FUNCTION_BLOCK FB_SequenceCONVEY_RETRACT EXTENDS FB_SequenceBase



VAR_IN_OUT
	devices: ST_POPComponents;
END_VAR

METHOD FB_init : BOOL
VAR_INPUT
	bInitRetains : BOOL; // if TRUE, the retain variables are initialized (warm start / cold start)
	bInCopyCode : BOOL;  // if TRUE, the instance afterwards gets moved into the copy code (online change)
	
	
END_VAR
(*
		Here we set the order of things to command, what the commands should be, and also how much time to allow during and between steps
		Every component listed below becomes 'Enabled' at each step
*)
sSequenceName:= 'POP Conveyor Reverse Sequence';
sSequenceDescription := 'Performs the full reverse series of actions (starting with lifting movement and followed by static conveyors';
bSequentional_1_Flood_0 := TRUE;
END_METHOD

METHOD populateSteps : ST_SequenceStep
VAR_INPUT
	
END_VAR
(*
		Here we set the order of things to command, what the commands should be, and also how much time to allow during and between steps
		Every component listed below becomes 'Enabled' at each step
*)

Step1.Device := devices.fbLinAct_POP1;
Step1.Command := E_DeviceState.RETRACTED;
Step1.StepMinDuration := T#0S; 
Step1.DelayUntilNextStep := T#0S;
Step1.WaitForAction := FALSE;
aSequenceSteps[1] :=   Step1;

Step2.Device := devices.fbLinAct_POP1;
Step2.Command := E_DeviceState.RETRACTED;
Step2.StepMinDuration := T#0S; 
Step2.DelayUntilNextStep := T#0S;
Step2.WaitForAction := FALSE;
aSequenceSteps[2] :=   Step2;

Step3.Device := devices.fbLinAct_POP2;
Step3.Command := E_DeviceState.RETRACTED;
Step3.StepMinDuration := T#0S;
Step3.DelayUntilNextStep := T#0S;
Step3.WaitForAction := FALSE;
aSequenceSteps[3] :=   Step3;

Step4.Device := devices.fbTrayCentre_POP1;
Step4.Command := E_DeviceState.RETRACTED;
Step4.StepMinDuration := T#0S;
Step4.DelayUntilNextStep := T#0S;
Step4.WaitForAction := FALSE;
aSequenceSteps[4] :=   Step4;

Step5.Device := devices.fbTrayCentre_POP2;
Step5.Command := E_DeviceState.RETRACTED;
Step5.StepMinDuration := T#0S;
Step5.DelayUntilNextStep := T#0S;
Step5.WaitForAction := FALSE;
aSequenceSteps[5] :=   Step5;

Step6.Device := devices.fbTrayCentre_POP3;
Step6.Command := E_DeviceState.RETRACTED;
Step6.StepMinDuration := T#0S;
Step6.DelayUntilNextStep := T#0S;
Step6.WaitForAction := FALSE;
aSequenceSteps[6] :=   Step6;

Step7.Device := devices.fbTrayEndSensor;
Step7.Command := E_DeviceState.ON;
Step7.StepMinDuration := T#0S;
Step7.DelayUntilNextStep := T#0S;
Step7.WaitForAction := TRUE;
aSequenceSteps[6] :=   Step7;


Step8.Device := devices.fbLinAct_POP1;
Step8.Command := E_DeviceState.EXTENDED;
Step8.StepMinDuration := T#0S;
Step8.DelayUntilNextStep := T#0S;
Step8.WaitForAction := FALSE;
aSequenceSteps[8] :=   Step8;

Step9.Device := devices.fbLinAct_POP2;
Step9.Command := E_DeviceState.EXTENDED;
Step9.StepMinDuration := T#0S;
Step9.DelayUntilNextStep := T#0S;
Step9.WaitForAction := FALSE;
aSequenceSteps[9] :=   Step9;

Step10.Device := devices.fbLinAct_POP3;
Step10.Command := E_DeviceState.EXTENDED;
Step10.StepMinDuration := T#0S;
Step10.DelayUntilNextStep := T#0S;
Step10.WaitForAction := TRUE;
aSequenceSteps[10] :=   Step10;

Step11.Device := devices.fbStaticConv_POP1;
Step11.Command := E_DeviceState.RUNNING;
Step11.StepMinDuration := T#0S; 
Step11.DelayUntilNextStep := T#0S;
Step11.WaitForAction := FALSE;
aSequenceSteps[11] :=   Step11;

Step12.Device := devices.fbStaticConv_POP2;
Step12.Command := E_DeviceState.RUNNING;
Step12.StepMinDuration := T#0S; 
Step12.DelayUntilNextStep := T#0S;
Step12.WaitForAction := FALSE;
aSequenceSteps[12] :=   Step12;

Step13.Device := devices.fbStaticConv_POP3;
Step13.Command := E_DeviceState.RUNNING;
Step13.StepMinDuration := T#0S; 
Step13.DelayUntilNextStep := T#0S;
Step13.WaitForAction := FALSE;
aSequenceSteps[13] :=   Step13;


Step14.Device := devices.fbTrayEndSensor;
Step14.Command := E_DeviceState.OFF;
Step14.StepMinDuration := T#0S; 
Step14.DelayUntilNextStep := T#0S;
Step14.WaitForAction := TRUE;
aSequenceSteps[14] :=   Step14;


nNumberSequenceSteps := 14;  // use this number to limit the number of operations
updateVarIDs();
END_METHOD

END_FUNCTION_BLOCK

(* stored: Version 1.1.0.1, ProductVersion 3.1.4024.12
   POU FB_SequenceCONVEY_RETRACT: Id {059b4c92-8bc2-4548-8bf6-1d5f50ffe4f6}, SpecialFunc None
   Method FB_init: Id {51382c7e-3456-4484-878f-c61dd0414672}
   Method populateSteps: Id {03fcd1db-d1b8-4f93-ae3c-5d101c486850} *)
